// TIA Portal V20 export
// export: Created 2026-07-10T11:12:28.0647884Z, ExportSetting WithDefaults, DisplayName Totally Integrated Automation Portal, DisplayVersion V20, DisplayName TIA Portal Openness, DisplayVersion V20, DisplayName TIA Portal Version Control Interface, DisplayVersion V20, DisplayName STEP 7 Professional, DisplayVersion V20, DisplayName STEP 7 Safety, DisplayVersion V20, DisplayName WinCC Basic/Comfort/Advanced, DisplayVersion V20, DisplayName WinCC Unified, DisplayVersion V20
DATA_BLOCK "MB_Config"   // DB14
{ S7_Optimized_Access := 'TRUE' }
VERSION : 0.1
// stored: AutoNumber true, DBAccessibleFromOPCUA true, IsOnlyStoredInLoadMemory false, IsRetainMemResEnabled false, IsWriteProtectedInAS false, MemoryReserve 100
   VAR
      CONNECT : TCON_IP_v4;
      NDR : Bool := FALSE;
      DR : Bool := FALSE;
      ERROR : Bool := FALSE;
      STATUS : Word := 16#0000;
      BUFFER : Array[0..500] of Word;
   END_VAR
BEGIN
   CONNECT.InterfaceId := 64;
   CONNECT.ID := 16#0001;
   CONNECT.ConnectionType := 16#0B;
   CONNECT.ActiveEstablished := FALSE;
   CONNECT.RemoteAddress.ADDR[1..4] := 16#00;
   CONNECT.RemotePort := 0;
   CONNECT.LocalPort := 502;
   BUFFER[0..500] := 16#0000;
END_DATA_BLOCK
